FUNCTION_BLOCK FB_TCPServer

VAR
	sLocalHost: T_IPv4Addr;
	nLocalPort: UDINT := 9000;
	//bStartCommunication : BOOL;
	sNetId	:T_AmsNetId;
	//bSent	: BOOL;

	bConnected: BOOL;
	sSendData: STRING(255);
	bBusy: BOOL;	
	bError: BOOL;
	nErrorID: UDINT;
	sDataRev: STRING(255);

	//iState: INT;
	hListener: T_HSOCKET;
	hSocket: T_HSOCKET;
	fbSocketAccept: FB_SocketAccept;
	fbSocketListen: FB_SocketListen;
	fbSocketReceive: FB_SocketReceive;
	fbSocketClose: FB_SocketClose;
	fbSocketCloseAll: FB_SocketCloseAll;
	fbSocketSend: FB_SocketSend;
	bAcceptExecute: BOOL;
	sReadData: STRING(255);
	ReceiveCounter: UDINT;
	bSocketCloseError: BOOL;
	nSocketCloseError: UDINT;
	//bSendTrigger: BOOL;
	//sData : STRING(255);
	iStepGeneral	: INT := 0;
	iStepStop		: INT := 0;
END_VAR

StateMachine();
IF bError THEN
	iStepGeneral := 50;
END_IF

METHOD Connect : BOOL
VAR_INPUT
END_VAR
IF NOT bConnected AND NOT bError THEN
	iStepGeneral := 1;
END_IF
END_METHOD

PROPERTY DataRev : String(255)
GET
DataRev := sDataRev;
END_GET
END_PROPERTY

METHOD Disconnect : BOOL
VAR_INPUT
END_VAR
iStepGeneral := 50;
END_METHOD

PROPERTY Error : bool
GET
Error	:= bError;
END_GET
END_PROPERTY

PROPERTY IsConnect : bool
GET
IsConnect	:= bConnected;
END_GET
END_PROPERTY

PROPERTY LocalHost : T_IPv4Addr
SET
sLocalHost	:= LocalHost;
END_SET
END_PROPERTY

PROPERTY LocalPort : UDINT
SET
//nLocalPort	:= LocalPort;
END_SET
END_PROPERTY

PROPERTY NetId : T_AmsNetId
SET
sNetId	:= NetId;
END_SET
END_PROPERTY

METHOD SendData : BOOL
VAR_INPUT
	DataSend	: STRING(255);
END_VAR
sSendData := DataSend;
IF bConnected OR bError THEN
	IF iStepGeneral = 30 THEN
		iStepGeneral := 40;
	END_IF
END_IF
END_METHOD

METHOD private StateAccept : BOOL
VAR_INPUT
END_VAR
fbSocketAccept(																
		sSrvNetId:= sNetId, 		
		hListener:= hListener, 													
		bExecute:= TRUE, 
		tTimeout:= T#4S, 
		bAccepted=> , 
		bBusy=> bBusy, 
		bError=> bError, 
		nErrId=> nErrorID,
		hSocket=> hSocket);														
	IF NOT fbSocketAccept.bBusy THEN
		fbSocketAccept(bExecute:= FALSE);
	END_IF

	IF bError THEN
		iStepGeneral := 50; 
	ELSIF hSocket.handle <> 0 THEN
		iStepGeneral := iStepGeneral + 10; 
		bConnected := TRUE;
	END_IF
END_METHOD

METHOD PRIVATE StateClose : BOOL
VAR_INPUT
END_VAR
CASE iStepStop OF
0:	// Error Handling	
	fbSocketClose(																// Close Listener-Socket
		sSrvNetId:= sNetId, 
		hSocket:= hListener, 
		bExecute:= TRUE, 
		tTimeout:= T#4S, 
		bBusy=> , 
		bError=> bError, 
		nErrId=> nErrorID);		
	IF (NOT fbSocketClose.bBusy) OR fbSocketClose.bError THEN
		hListener.handle := 0;
		iStepStop := iStepStop + 1;
	END_IF
1:	
	fbSocketClose(bExecute := FALSE);
	iStepStop := iStepStop + 1;
2:
	fbSocketClose(																// Close Connection Socket
		sSrvNetId:= sNetId, 
		hSocket:= hSocket, 
		bExecute:= TRUE, 
		tTimeout:= T#4S, 
		bBusy=> , 
		bError=> bError, 
		nErrId=> nErrorID);
	IF NOT (fbSocketClose.bBusy) OR fbSocketClose.bError THEN
		hSocket.handle 	:= 0;	
		iStepGeneral 	:= 0;
		iStepStop		:= 0;
		bConnected 		:= FALSE;
	END_IF
END_CASE
END_METHOD

METHOD PRIVATE StateInit : BOOL
VAR_INPUT
END_VAR
fbSocketCloseAll(
		sSrvNetId:= sNetId, 
		bExecute:= TRUE, 
		tTimeout:= T#3S, 
		bBusy=> , 
		bError=> bSocketCloseError, 
		nErrId=> nSocketCloseError);

IF NOT (fbSocketCloseAll.bBusy OR fbSocketCloseAll.bError) THEN
		fbSocketCloseAll(bExecute:= FALSE);
		fbSocketListen(bExecute := FALSE);
		fbSocketAccept(bExecute := FALSE);
		fbSocketClose(bExecute:= FALSE);
		bConnected	:= FALSE;
		bBusy 		:= TRUE;
		iStepGeneral := 10;
END_IF
END_METHOD

METHOD PRIVATE StateListen : BOOL
VAR_INPUT
END_VAR
fbSocketListen(																
		sSrvNetId:= sNetId, 														
		sLocalHost:= sLocalHost, 												
		nLocalPort:= nLocalPort, 												
		bExecute:= TRUE, 
		tTimeout:= T#4S, 
		bBusy=> bBusy, 
		bError=> bError, 
		nErrId=> nErrorID,
		hListener=> hListener);													
		
	IF hListener.handle <> 0 THEN
		iStepGeneral := iStepGeneral + 10;	
	ELSIF bError THEN
		iStepGeneral := 50;
	END_IF
END_METHOD

METHOD PRIVATE StateMachine : BOOL
VAR_INPUT
END_VAR
CASE iStepGeneral OF
	1:
		StateInit();
	10:
		StateListen();
	20:
		StateAccept();
	30:
		StateReceive();
	40:
		StateSend();
	50:
		StateClose();
END_CASE
END_METHOD

METHOD PRIVATE StateReceive : BOOL
VAR_INPUT
END_VAR
fbSocketReceive(															
		sSrvNetId:= sNetId, 
		hSocket:= hSocket, 
		cbLen:= SIZEOF(sReadData) , 
		pDest:= ADR(sReadData), 
		bExecute:= TRUE, 														
		tTimeout:= T#4S, 
		bBusy=> , 
		bError=> bError, 
		nErrId=> nErrorID,
		nRecBytes=> );
		
	IF NOT fbSocketReceive.bBusy THEN
		fbSocketReceive(bExecute := FALSE);
		IF fbSocketReceive.nRecBytes <> 0 THEN									
			sDataRev := sReadData;
		END_IF
	END_IF
	
	IF fbSocketReceive.bError OR(NOT bConnected) THEN					
		iStepGeneral := 50;
	END_IF
END_METHOD

METHOD PRIVATE StateSend : BOOL
VAR_INPUT
END_VAR
fbSocketSend(																// Send Data to client
		sSrvNetId:= sNetId, 
		hSocket:= hSocket, 
		cbLen:= SIZEOF(sSendData), 
		pSrc:= ADR(sSendData),
		bExecute:= TRUE, 
		tTimeout:= T#3S, 
		bBusy=> , 
		bError=> bError, 
		nErrId=> nErrorID);	
	
	IF NOT fbSocketSend.bBusy THEN												// Switch back to receiving state after sending
		iStepGeneral := iStepGeneral - 10;
	ELSIF fbSocketSend.bError OR NOT bConnected THEN
		iStepGeneral := 50;													// Close connection in case of error 
	END_IF
END_METHOD

END_FUNCTION_BLOCK

(* stored: Version 1.1.0.1, ProductVersion 3.1.4024.12
   POU FB_TCPServer: Id {eaed78c2-34d1-42b7-98f4-b58fa196fe7c}, SpecialFunc None
   Folder Property: Id {f144cff3-1a2d-40e7-a2ed-669d7ab1a02b}
   Folder Request: Id {54531ff0-b064-45c7-8196-eb2a931fdd5e}
   Folder StateMachine: Id {eebc7770-41d7-4656-97ea-5def8c1a255f}
   Method Connect: Id {f07c0af8-fe4f-482b-979b-a526c29434e2}
   Property DataRev: Id {a4e638e6-dfa1-4334-8209-4437e9039d14}
   Get Get: Id {a35e3adc-26a1-472a-8847-1fa1686c7b20}
   Method Disconnect: Id {f3511e92-12fb-44f7-9c4d-2714d7fb6c9a}
   Property Error: Id {7a447f67-3aea-4771-885d-4aa07b8a93fb}
   Get Get: Id {c30990f4-29b5-47e2-a796-4aae3640f023}
   Property IsConnect: Id {90545187-2ecb-4d38-830c-212af879abe7}
   Get Get: Id {f4af79a5-76e2-41f6-ba73-704899e2c4a2}
   Property LocalHost: Id {4b14a993-dad8-4a02-b6dc-e308d885d81e}
   Set Set: Id {7db50b28-a2fe-4dcc-bb68-d0f22f7c4718}
   Property LocalPort: Id {ba9111b5-c1a2-44e4-9320-9537312776fc}
   Set Set: Id {b5c21f53-f9e8-4751-a7dd-97917c177d8d}
   Property NetId: Id {61d3a761-ba5b-48f1-99f1-825ea1c9a015}
   Set Set: Id {54e00d8b-840c-4594-8efb-094568e2f230}
   Method SendData: Id {b0a31b62-31ab-46c3-aa23-15c0d0113e3b}
   Method StateAccept: Id {e54edb93-e854-4dd5-9adc-480d46711809}
   Method StateClose: Id {2a5e788a-4a9d-4455-850d-8be8c7890e72}
   Method StateInit: Id {c86ea60a-26db-47e4-b0e1-923e6e65d646}
   Method StateListen: Id {87f37b74-b72a-4c99-85ba-a1d4657fa90b}
   Method StateMachine: Id {53701d1c-8d46-47b7-b412-3534c3493e1e}
   Method StateReceive: Id {d037dafd-38a5-406d-bbaf-d37dbd38c180}
   Method StateSend: Id {0ec2b539-7683-4687-a5e4-0314df51f7b8} *)
